{attribute 'GeneratedUsingTerminal: EL9182--0000'}
{attribute addProperty BoxType "EL9182--0000"}
{attribute addProperty Description "EL9182 Potential Connection, 8 x 2 contacts"}
{attribute addProperty Physics "KK"}
{attribute addProperty Id "EL9182"}
{attribute addProperty CRC "2190947810"}
{attribute addProperty Size "0"}
TYPE EL9182_829735E2 EXTENDS EtcSlaveTerminalBase_947E5A46 :
STRUCT
END_STRUCT
END_TYPE

(* stored: Version 1.2.0.0, ProductVersion 3.1.4024.11
   DUT EL9182_829735E2: Id {e8f076e2-2608-4916-91c7-0be001133ceb} *)
